FUNCTION_BLOCK FB_Axis_1
VAR_INPUT
	sAxis_Name		: STRING:='Axis Name';	
	bSen_Homming	: BOOL;
	eHomeMode		: MC_HomingMode:=MC_HomingMode.MC_Direct;
	eAxis_Name		: E_Axis_Name;




END_VAR
VAR_OUTPUT
END_VAR
VAR
	Axis			: REFERENCE TO ST_Axis;
	Axis_ref		: REFERENCE TO AXIS_REF;	
	sAxis_Num		: INT;

	mcPower			: MC_Power;
	mcReset			: MC_Reset;
	mcSetPosition	: MC_SetPosition;
	mcMoveAbs		: MC_MoveAbsolute;
	mcMoveAbs2		: MC_MoveAbsolute;
	mcMoveRel		: MC_MoveRelative;
	mcMoveRel2		: MC_MoveRelative;
	mcMoveMod		: MC_MoveModulo;
	mcMoveMod2		: MC_MoveModulo;
	mcMoveVel		: MC_MoveVelocity;
	mcHome			: MC_Home;


	
	mcStop			: MC_Stop;
	mcJog			: MC_Jog;
	
	ReadSdo					: FB_EcCoESdoRead;
	nIndexErrorSOD			: WORD:=16#603F;//h
	iErrorDI				: WORD;
	pError					: POINTER TO BYTE :=ADR(iErrorDI);
	bReadError				: BOOL;
	rt_ReadDriveError		: R_TRIG;
	ft_ReadDriveError		: F_TRIG;
	
	
	ton_Reset: TON;
END_VAR
VAR_IN_OUT

END_VAR

act_Get_Reference();
AXIS_REF.ReadStatus();
Axis.sAxis_Name:=sAxis_Name;
Axis.sAxis_Num:=sAxis_Num:=eAxis_Name;

Axis.bEnabled:=NOT AXIS_REF.Status.Disabled AND AXIS_REF.Status.Operational;
Axis.bError:=AXIS_REF.Status.Error;
Axis.bHomeSen:=bSen_Homming;
Axis.bHomeDone:=AXIS_REF.Status.Homed;
Axis.eHomeMode:=eHomeMode;
act_Call_Function();

Axis.fActPos:=Axis_ref.NcToPlc.ActPos;
Axis.fActPosModulo:=Axis_ref.NcToPlc.ModuloActPos;

Axis.fActVelo:=Axis_ref.NcToPlc.ActVelo;

act_Read_Error_SDO();
Axis.iErrorDI:=iErrorDI;

ACTION act_Call_Function:
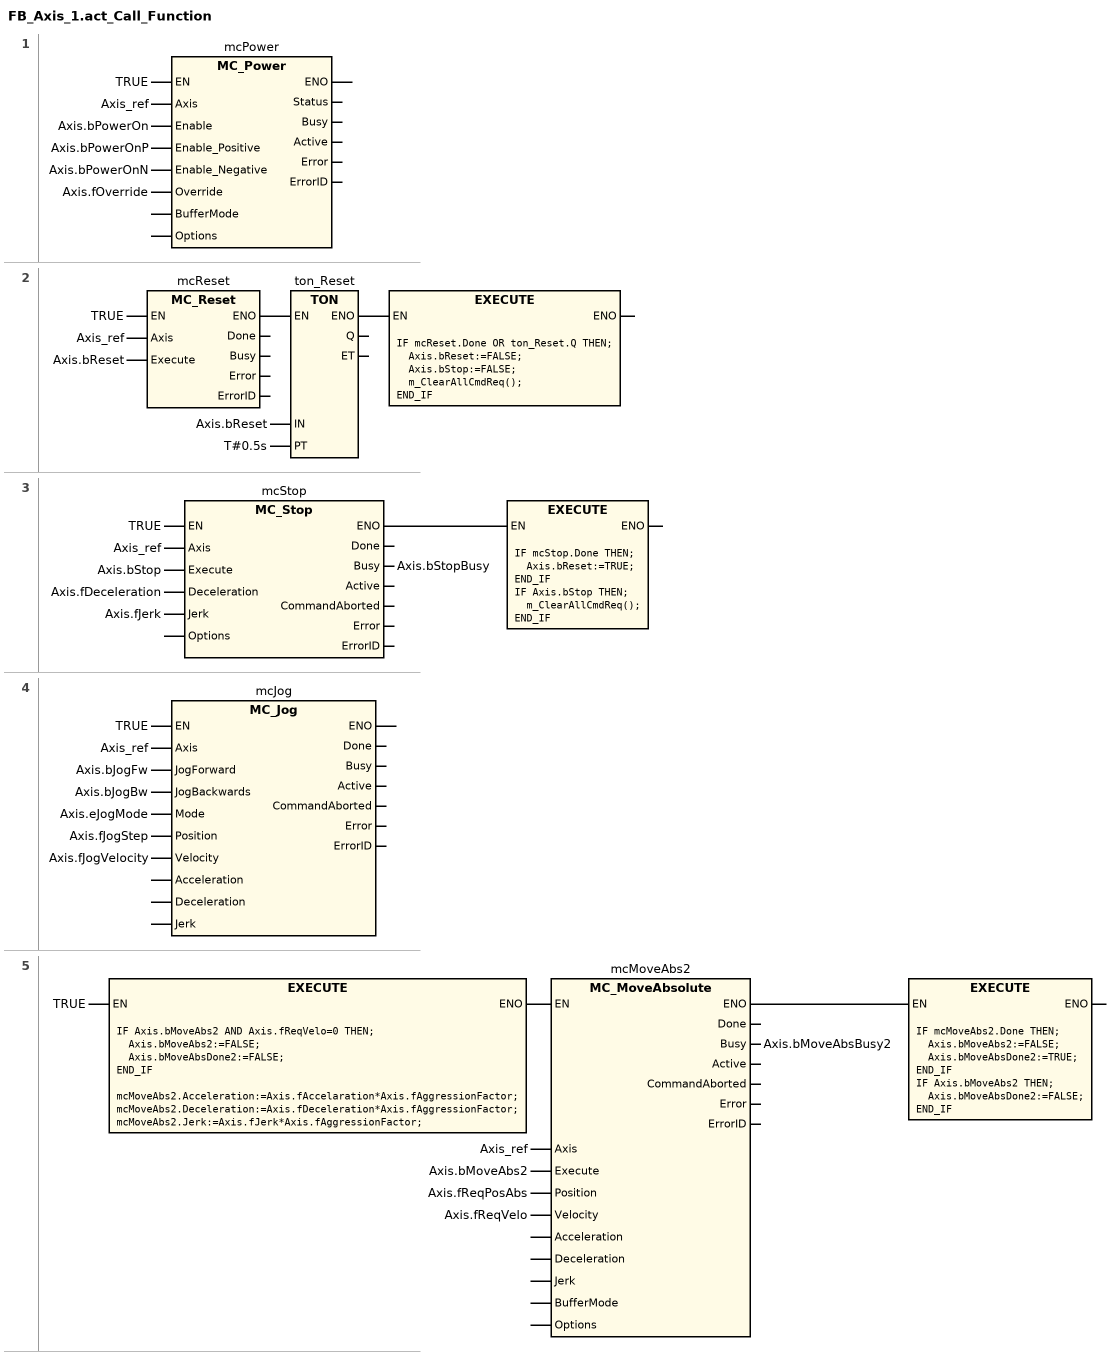
// NETWORK 1
mcPower(
    Axis := Axis_ref,
    Enable := Axis.bPowerOn,
    Enable_Positive := Axis.bPowerOnP,
    Enable_Negative := Axis.bPowerOnN,
    Override := Axis.fOverride); // MC_Power

// NETWORK 2
mcReset(Axis := Axis_ref, Execute := Axis.bReset); // MC_Reset
ton_Reset(IN := Axis.bReset, PT := T#0.5s); // TON

IF mcReset.Done OR ton_Reset.Q THEN;
	Axis.bReset:=FALSE;
	Axis.bStop:=FALSE;
	m_ClearAllCmdReq();
END_IF

// NETWORK 3
mcStop(
    Axis := Axis_ref,
    Execute := Axis.bStop,
    Deceleration := Axis.fDeceleration,
    Jerk := Axis.fJerk,
    Busy => Axis.bStopBusy); // MC_Stop

IF mcStop.Done THEN;
	Axis.bReset:=TRUE;
END_IF
IF Axis.bStop THEN;
	m_ClearAllCmdReq();
END_IF

// NETWORK 4
mcJog(
    Axis := Axis_ref,
    JogForward := Axis.bJogFw,
    JogBackwards := Axis.bJogBw,
    Mode := Axis.eJogMode,
    Position := Axis.fJogStep,
    Velocity := Axis.fJogVelocity); // MC_Jog

// NETWORK 5

IF Axis.bMoveAbs2 AND Axis.fReqVelo=0 THEN;
	Axis.bMoveAbs2:=FALSE;
	Axis.bMoveAbsDone2:=FALSE;
END_IF

mcMoveAbs2.Acceleration:=Axis.fAccelaration*Axis.fAggressionFactor;
mcMoveAbs2.Deceleration:=Axis.fDeceleration*Axis.fAggressionFactor;
mcMoveAbs2.Jerk:=Axis.fJerk*Axis.fAggressionFactor;
mcMoveAbs2(
    Axis := Axis_ref,
    Execute := Axis.bMoveAbs2,
    Position := Axis.fReqPosAbs,
    Velocity := Axis.fReqVelo,
    Busy => Axis.bMoveAbsBusy2); // MC_MoveAbsolute

IF mcMoveAbs2.Done THEN;
	Axis.bMoveAbs2:=FALSE;
	Axis.bMoveAbsDone2:=TRUE;
END_IF
IF Axis.bMoveAbs2 THEN;
	Axis.bMoveAbsDone2:=FALSE;
END_IF

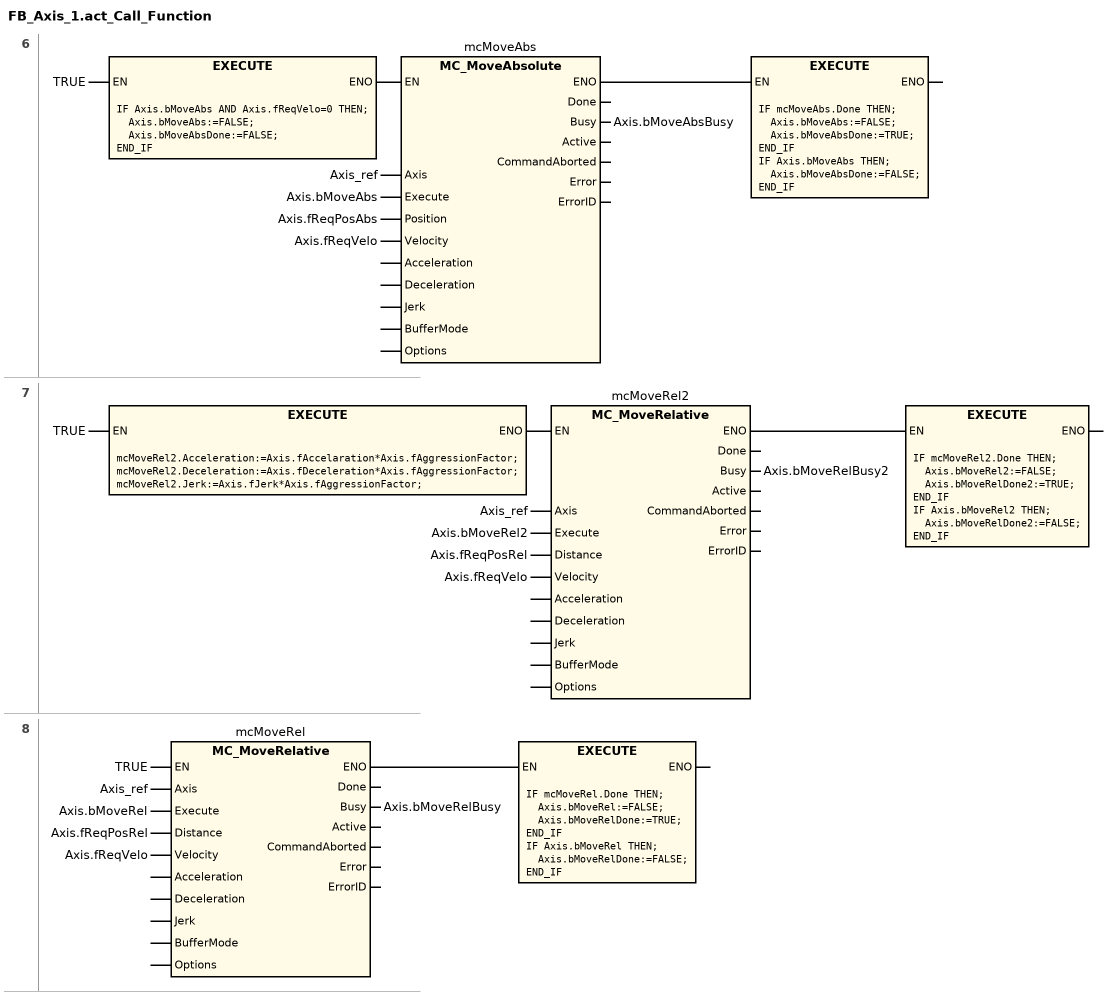
// NETWORK 6

IF Axis.bMoveAbs AND Axis.fReqVelo=0 THEN;
	Axis.bMoveAbs:=FALSE;
	Axis.bMoveAbsDone:=FALSE;
END_IF
mcMoveAbs(
    Axis := Axis_ref,
    Execute := Axis.bMoveAbs,
    Position := Axis.fReqPosAbs,
    Velocity := Axis.fReqVelo,
    Busy => Axis.bMoveAbsBusy); // MC_MoveAbsolute

IF mcMoveAbs.Done THEN;
	Axis.bMoveAbs:=FALSE;
	Axis.bMoveAbsDone:=TRUE;
END_IF
IF Axis.bMoveAbs THEN;
	Axis.bMoveAbsDone:=FALSE;
END_IF

// NETWORK 7

mcMoveRel2.Acceleration:=Axis.fAccelaration*Axis.fAggressionFactor;
mcMoveRel2.Deceleration:=Axis.fDeceleration*Axis.fAggressionFactor;
mcMoveRel2.Jerk:=Axis.fJerk*Axis.fAggressionFactor;
mcMoveRel2(
    Axis := Axis_ref,
    Execute := Axis.bMoveRel2,
    Distance := Axis.fReqPosRel,
    Velocity := Axis.fReqVelo,
    Busy => Axis.bMoveRelBusy2); // MC_MoveRelative

IF mcMoveRel2.Done THEN;
	Axis.bMoveRel2:=FALSE;
	Axis.bMoveRelDone2:=TRUE;
END_IF
IF Axis.bMoveRel2 THEN;
	Axis.bMoveRelDone2:=FALSE;
END_IF

// NETWORK 8
mcMoveRel(
    Axis := Axis_ref,
    Execute := Axis.bMoveRel,
    Distance := Axis.fReqPosRel,
    Velocity := Axis.fReqVelo,
    Busy => Axis.bMoveRelBusy); // MC_MoveRelative

IF mcMoveRel.Done THEN;
	Axis.bMoveRel:=FALSE;
	Axis.bMoveRelDone:=TRUE;
END_IF
IF Axis.bMoveRel THEN;
	Axis.bMoveRelDone:=FALSE;
END_IF

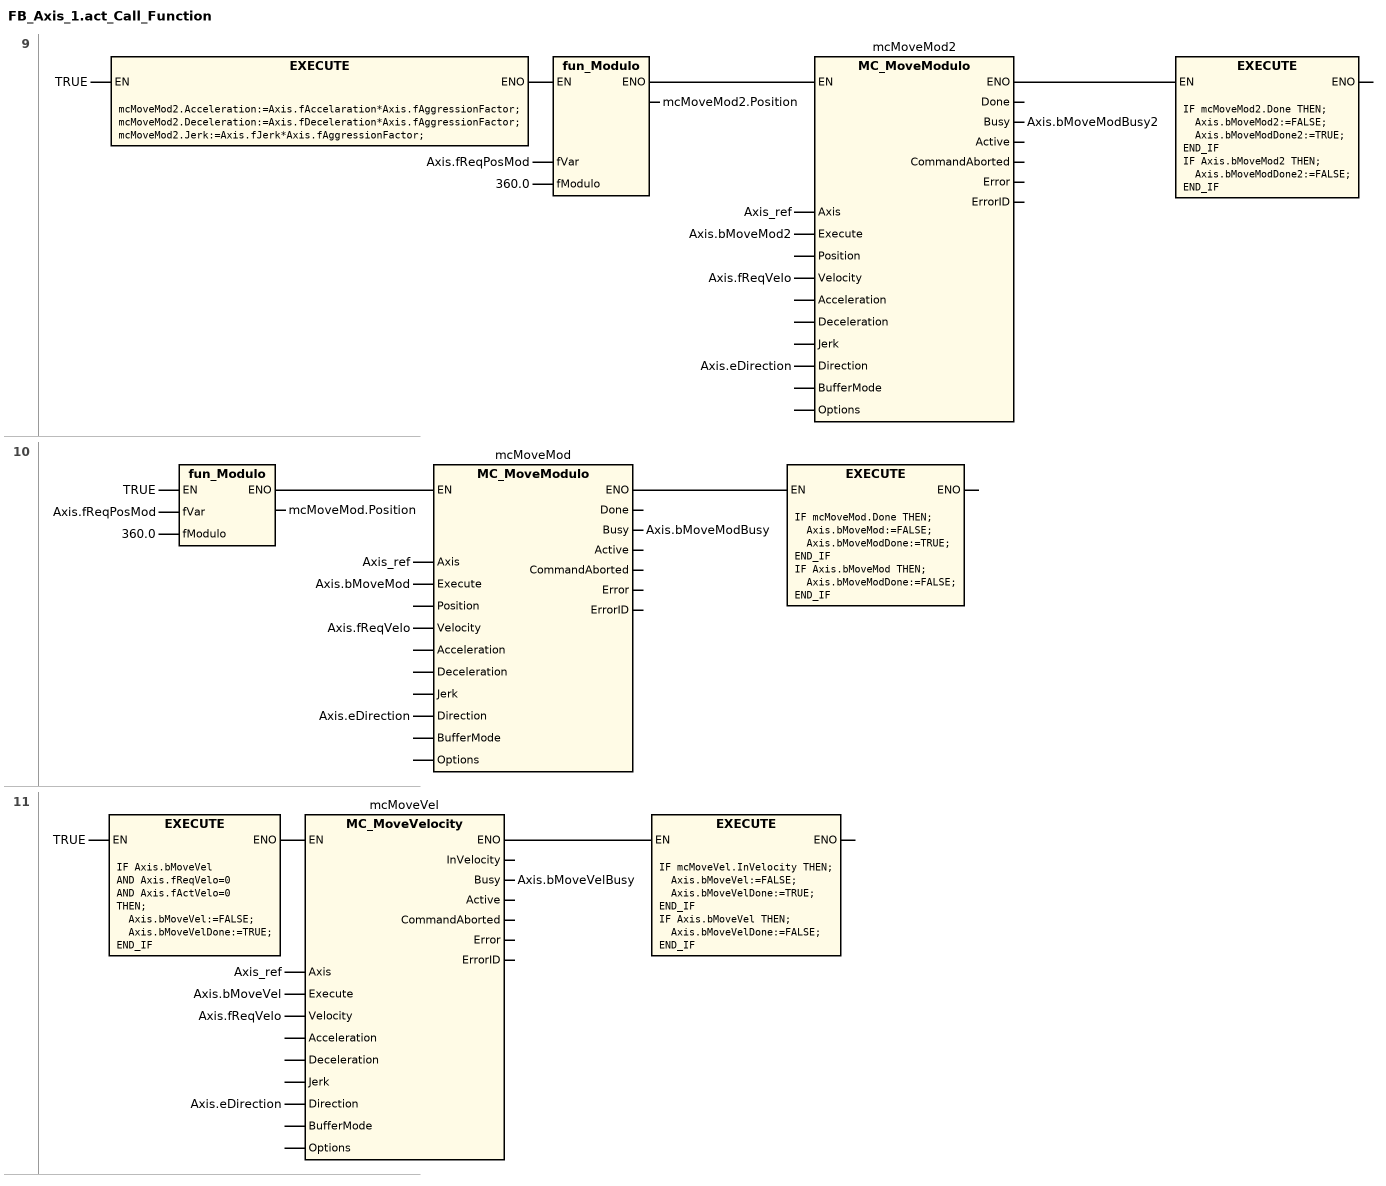
// NETWORK 9

mcMoveMod2.Acceleration:=Axis.fAccelaration*Axis.fAggressionFactor;
mcMoveMod2.Deceleration:=Axis.fDeceleration*Axis.fAggressionFactor;
mcMoveMod2.Jerk:=Axis.fJerk*Axis.fAggressionFactor;
mcMoveMod2.Position := fun_Modulo(fVar := Axis.fReqPosMod, fModulo := 360.0);
mcMoveMod2(
    Axis := Axis_ref,
    Execute := Axis.bMoveMod2,
    Velocity := Axis.fReqVelo,
    Direction := Axis.eDirection,
    Busy => Axis.bMoveModBusy2); // MC_MoveModulo

IF mcMoveMod2.Done THEN;
	Axis.bMoveMod2:=FALSE;
	Axis.bMoveModDone2:=TRUE;
END_IF
IF Axis.bMoveMod2 THEN;
	Axis.bMoveModDone2:=FALSE;
END_IF

// NETWORK 10
mcMoveMod.Position := fun_Modulo(fVar := Axis.fReqPosMod, fModulo := 360.0);
mcMoveMod(
    Axis := Axis_ref,
    Execute := Axis.bMoveMod,
    Velocity := Axis.fReqVelo,
    Direction := Axis.eDirection,
    Busy => Axis.bMoveModBusy); // MC_MoveModulo

IF mcMoveMod.Done THEN;
	Axis.bMoveMod:=FALSE;
	Axis.bMoveModDone:=TRUE;
END_IF
IF Axis.bMoveMod THEN;
	Axis.bMoveModDone:=FALSE;
END_IF

// NETWORK 11

IF Axis.bMoveVel 
AND Axis.fReqVelo=0 
AND Axis.fActVelo=0
THEN;
	Axis.bMoveVel:=FALSE;
	Axis.bMoveVelDone:=TRUE;
END_IF
mcMoveVel(
    Axis := Axis_ref,
    Execute := Axis.bMoveVel,
    Velocity := Axis.fReqVelo,
    Direction := Axis.eDirection,
    Busy => Axis.bMoveVelBusy); // MC_MoveVelocity

IF mcMoveVel.InVelocity THEN;
	Axis.bMoveVel:=FALSE;
	Axis.bMoveVelDone:=TRUE;
END_IF
IF Axis.bMoveVel THEN;
	Axis.bMoveVelDone:=FALSE;
END_IF

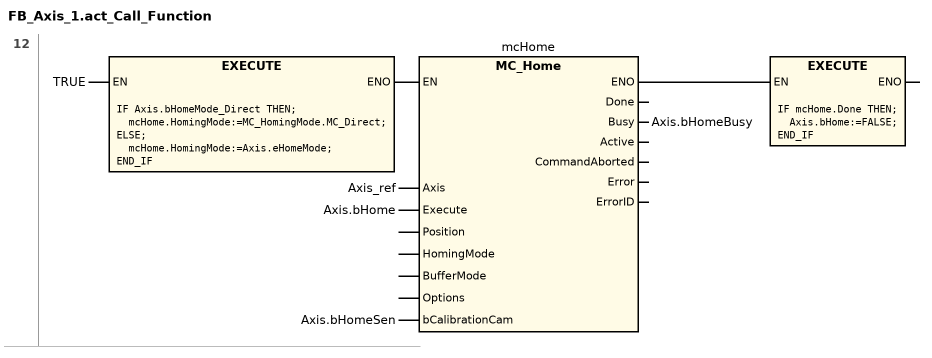
// NETWORK 12

IF Axis.bHomeMode_Direct THEN;
	mcHome.HomingMode:=MC_HomingMode.MC_Direct;
ELSE;
	mcHome.HomingMode:=Axis.eHomeMode;
END_IF
mcHome(Axis := Axis_ref, Execute := Axis.bHome, bCalibrationCam := Axis.bHomeSen, Busy => Axis.bHomeBusy); // MC_Home

IF mcHome.Done THEN;
	Axis.bHome:=FALSE;
END_IF
END_ACTION

ACTION act_Get_Reference:
Axis REF= g_Axis.stAxis[eAxis_Name];
Axis_ref REF= g_Axis.AxisRef[eAxis_Name];
Axis.Status REF= Axis_ref.Status;
END_ACTION

ACTION act_Read_Error_SDO:
rt_ReadDriveError(CLK:=Axis_ref.Status.Error);
ft_ReadDriveError(CLK:=Axis_ref.Status.Error);

IF 	rt_ReadDriveError.Q OR ft_ReadDriveError.Q THEN;
	bReadError:=TRUE;
END_IF

ReadSdo(
	sNetId:= F_CreateAmsNetId(g_in.adrDrive_AMS_Info[eAxis_Name].netId), 
	nSlaveAddr:= g_in.adrDrive_AMS_Info[eAxis_Name].port, 
	nSubIndex:= , 
	nIndex:= nIndexErrorSOD, 
	pDstBuf:= pError, 
	cbBufLen:= 2, 
	bExecute:= bReadError, 
	tTimeout:= , 
	bBusy=> , 
	bError=> , 
	nErrId=> , 
	cbRead=> );

bReadError:=FALSE;
iErrorDI;
END_ACTION

METHOD m_ClearAllCmdReq : BOOL
VAR_INPUT
END_VAR
Axis.bJogFw :=Axis.bJogBw :=Axis.bHome  :=FALSE;
Axis.bMoveAbsDone :=Axis.bMoveAbs :=FALSE;
Axis.bMoveAbsDone2:=Axis.bMoveAbs2:=FALSE;	
Axis.bMoveRelDone :=Axis.bMoveRel :=FALSE;
Axis.bMoveRelDone2:=Axis.bMoveRel2:=FALSE;	
Axis.bMoveModDone :=Axis.bMoveMod :=FALSE;
Axis.bMoveModDone2:=Axis.bMoveMod2:=FALSE;
Axis.bMoveVelDone :=Axis.bMoveVel :=FALSE;
END_METHOD

END_FUNCTION_BLOCK

(* stored: Version 1.1.0.1, ProductVersion 3.1.4024.12
   POU FB_Axis_1: Id {f3f2e80d-94ef-428f-b3f9-eead34e9e273}, SpecialFunc None
   Action act_Call_Function: Id {0b7cbafe-d4cd-4d19-b1c4-490dee63febb}
   Action act_Get_Reference: Id {51958983-d6d7-45d3-a558-ce5426bc2e24}
   Action act_Read_Error_SDO: Id {a6c65c01-f54a-4596-9e3b-79ffb41d3c99}
   Method m_ClearAllCmdReq: Id {b620ffea-b891-4625-b050-e8c259b5d2a7} *)
